(* IEC 61131-3 sources: plc_generation_empirical_study/datasets/task_bank_c06_bounded_runtime_v0_2/tasks/C06_R10_lean_composite, 2 files *)

(* ---- interface.st ---- *)
FUNCTION_BLOCK C06_R10_lean_composite
VAR_INPUT
    A_Inspected : BOOL;
    A_Rejected : BOOL;
    A_Reset : BOOL;
    A_WindowSize : INT;
    A_RejectLimit : INT;
    B_Ch1 : BOOL;
    B_Ch2 : BOOL;
    B_Ch3 : BOOL;
    B_AutoMode : BOOL;
    B_AutoRequest : BOOL;
    B_ManualRequest : BOOL;
    B_BypassRequest : BOOL;
    B_BypassPermit : BOOL;
    B_SafetyOK : BOOL;
    B_Reset : BOOL;
    SubsystemBEnable : BOOL;
    CrossReset : BOOL;
END_VAR
VAR_OUTPUT
    A_WindowCount : INT;
    A_RejectCount : INT;
    A_LockedOut : BOOL;
    A_WindowComplete : BOOL;
    B_RunPermit : BOOL;
    B_Degraded : BOOL;
    B_BypassActive : BOOL;
    B_Blocked : BOOL;
    CrossReady : BOOL;
    CrossBlocked : BOOL;
END_VAR
END_FUNCTION_BLOCK

(* ---- reference.st ---- *)
FUNCTION_BLOCK C06_R10_lean_composite
VAR_INPUT
    A_Inspected : BOOL;
    A_Rejected : BOOL;
    A_Reset : BOOL;
    A_WindowSize : INT;
    A_RejectLimit : INT;
    B_Ch1 : BOOL;
    B_Ch2 : BOOL;
    B_Ch3 : BOOL;
    B_AutoMode : BOOL;
    B_AutoRequest : BOOL;
    B_ManualRequest : BOOL;
    B_BypassRequest : BOOL;
    B_BypassPermit : BOOL;
    B_SafetyOK : BOOL;
    B_Reset : BOOL;
    SubsystemBEnable : BOOL;
    CrossReset : BOOL;
END_VAR
VAR_OUTPUT
    A_WindowCount : INT;
    A_RejectCount : INT;
    A_LockedOut : BOOL;
    A_WindowComplete : BOOL;
    B_RunPermit : BOOL;
    B_Degraded : BOOL;
    B_BypassActive : BOOL;
    B_Blocked : BOOL;
    CrossReady : BOOL;
    CrossBlocked : BOOL;
END_VAR
VAR
    A_PrevInspected : BOOL := FALSE;
    B_SelectedRequest : BOOL;
    B_VoteOK : BOOL;
    B_AnyChannel : BOOL;
    B_Unanimous : BOOL;
END_VAR

A_WindowComplete := FALSE;
IF A_Reset THEN
    A_WindowCount := 0;
    A_RejectCount := 0;
    A_LockedOut := FALSE;
ELSIF (NOT A_LockedOut) AND A_Inspected AND (NOT A_PrevInspected) THEN
    A_WindowCount := A_WindowCount + 1;
    IF A_Rejected THEN
        A_RejectCount := A_RejectCount + 1;
    END_IF;
    IF A_WindowCount >= A_WindowSize THEN
        IF A_RejectCount > A_RejectLimit THEN
            A_LockedOut := TRUE;
        END_IF;
        A_WindowCount := 0;
        A_RejectCount := 0;
        A_WindowComplete := TRUE;
    END_IF;
END_IF;
A_PrevInspected := A_Inspected;

IF CrossReset THEN
    CrossReady := FALSE;
ELSIF A_LockedOut THEN
    CrossReady := TRUE;
END_IF;
CrossBlocked := SubsystemBEnable AND (NOT CrossReady);

IF SubsystemBEnable AND CrossReady THEN
    B_SelectedRequest := (B_AutoMode AND B_AutoRequest) OR ((NOT B_AutoMode) AND B_ManualRequest);
    B_VoteOK := (B_Ch1 AND B_Ch2) OR (B_Ch1 AND B_Ch3) OR (B_Ch2 AND B_Ch3);
    B_AnyChannel := B_Ch1 OR B_Ch2 OR B_Ch3;
    B_Unanimous := (B_Ch1 AND B_Ch2 AND B_Ch3) OR ((NOT B_Ch1) AND (NOT B_Ch2) AND (NOT B_Ch3));
    IF B_Reset AND (NOT B_AutoRequest) AND (NOT B_ManualRequest) THEN
        B_BypassActive := FALSE;
    ELSIF (NOT B_AutoMode) AND B_BypassRequest AND B_BypassPermit AND B_SafetyOK AND B_AnyChannel THEN
        B_BypassActive := TRUE;
    END_IF;
    B_RunPermit := B_SelectedRequest AND B_SafetyOK AND (B_VoteOK OR B_BypassActive);
    B_Degraded := B_RunPermit AND ((NOT B_Unanimous) OR B_BypassActive);
    B_Blocked := B_SelectedRequest AND (NOT B_RunPermit);
ELSE
    B_RunPermit := FALSE;
    B_Degraded := FALSE;
    B_BypassActive := FALSE;
    B_Blocked := FALSE;
END_IF;

END_FUNCTION_BLOCK
